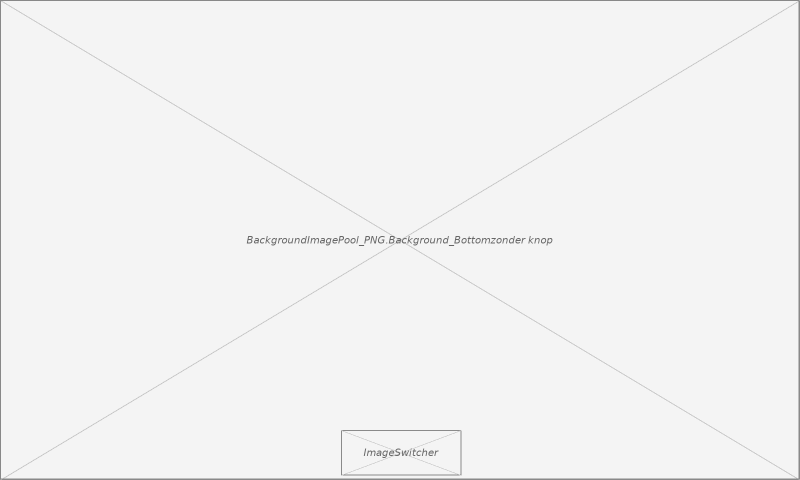
VISUALIZATION BackgroundNoButton  // 800x480
VAR_INPUT
	bHideEstop 			: BOOL ; // Hide emergency stop screen
	bDisableSettings	: BOOL ; // Deactivate settings
END_VAR
VAR_IN_OUT
	bCmdSettings	: BOOL ; // go to settings screen command
END_VAR
    Image (0,0 800x480), invisible if: bHideEstop, input disabled if: bHideEstop, image: BackgroundImagePool_PNG.Emergency Stop Active
    Image (0,0 800x480), image: BackgroundImagePool_PNG.Background_Bottomzonder knop
    ImageSwitcher (341,430 120x45), variable: GVL_HMI.bCmdSettings, input disabled if: bDisableSettings, background image: Buttons_PNG.Home-Settings Switch Pushed, image: Buttons_PNG.Home-Settings Switch, behaviour: TOGGLE
        p3148411668: Buttons_PNG.Home-Settings Switch Pushed
END_VISUALIZATION

(* stored: Version 1.1.0.1, ProductVersion 3.1.4024.11
   Visu BackgroundNoButton: Id {7b934ca9-86fe-4224-81d7-f07b866cae24} *)
